INTERFACE I_EncodedDrive EXTENDS I_PositionalDrive, I_ContinuousDrive
//this drive can perform absolute/relative targeting and continuous motion
//only used if a drive with both encoded and continuous behavior is needed

END_INTERFACE

(* stored: Version 1.1.0.1, ProductVersion 3.1.4024.11
   Itf I_EncodedDrive: Id {e1c482e6-9167-41ba-b08c-5b6653eac9da} *)
